(* CODESYS project codesysTest

Project tree, tasks and I/O mapping:
  Device : CODESYS Softmotion RTE V3 x64, 3S - Smart Software Solutions GmbH, version 3.5.18.30
    application Application
      libraries: Standard, 3.5.18.0 (System)
      task MainTask (cyclic, interval t#4ms, priority 1) calls PLC_PRG
      program PLC_PRG [ST]
    SoftMotion General Axis Pool
*)

// Device/Application/PLC_PRG
PROGRAM PLC_PRG
VAR
	i : UINT;
END_VAR

i:= i + 1;

END_PROGRAM
